// TIA Portal V19 export
TYPE "LAF_typePlasticRollerEm6ParametersInterfaceHmi"
// stored: Access Published
   STRUCT
      configuration : "LAF_typeRollerEm1ParametersHmi";
      commands : "LBC_typeInterfaceCommands";
      monitoring { S7_SetPoint := 'True'} : "LAF_typePlasticRollerEm6ProcessValuesHmi";
   END_STRUCT;
END_TYPE
